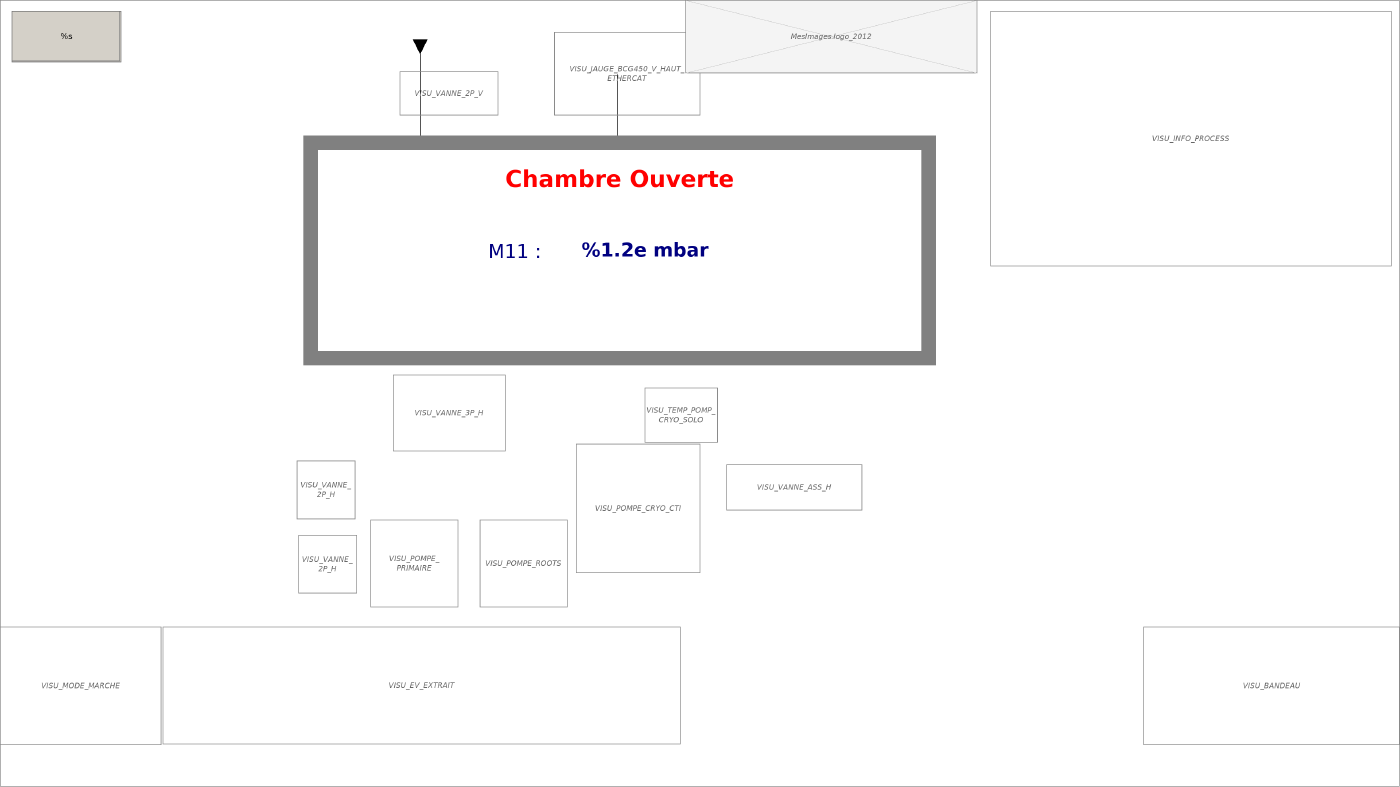
VISUALIZATION SYN_POMPAGE  // 1920x1080, background image fond_blanc_1280_1024
    Frame (223,860 710x161)
        shows VISU_EV_EXTRAIT()
    Frame (1568,860 352x162)
        shows VISU_BANDEAU(m_Input_MACHINE := Global_Variables.MACHINE)
    Frame (0,860 221x162)
        shows VISU_MODE_MARCHE(m_Input_MACHINE := .MACHINE)
    Button (16,15 150x70), "%s", text list: 'TextList_Navigation', text index: 1
        OnMouseClick: change screen: SYN_PROC
    Line (846,102) (846,217)
    Line (576,62) (576,216)
    RoundedRectangle (416,186 867x315)
    Frame (760,44 200x114)
        shows VISU_JAUGE_BCG450_V_HAUT_ETHERCAT(m_Input_JAUGE := PRG_POMPAGE.M11)
    Frame (548,98 135x60)
        shows VISU_VANNE_2P_V(m_Input_VANNE := PRG_POMPAGE.POMPAGE.VH11)
    Polygon (566,54) (586,54) (576,74)
    Rectangle (666,325 80x40), "M11 :"
    Rectangle (760,323 250x40), "%1.2e mbar", text variable: Global_Variables.PRG_POMPAGE.M11.STATE_Pression
    Label (669,214 362x63), "Chambre Ouverte", invisible if: PRG_POMPAGE.IN_FE11T
    Frame (1358,15 550x350), invisible if: NOT Global_Variables.MACHINE.STATE_Prod
        shows VISU_INFO_PROCESS()
    Polyline (458,705)
    Polyline (330,705)
    Polygon (337,745)
    Frame (407,632 80x80)
        shows VISU_VANNE_2P_H(m_Input_VANNE := PRG_POMPAGE.POMPAGE.VINT)
    Polyline (840,705)
    Frame (790,609 170x177)
        shows VISU_POMPE_CRYO_CTI(m_Input_POMPE := PRG_POMPAGE.POMPAGE.PS11, m_Input_COM := PRG_POMPAGE.COM_CRYOS, m_Input_Forcage := PRG_POMPAGE.POMPAGE.PS11.PRM_Forcage_Cryo_EXT)
    Polyline (553,751)
    Frame (884,532 100x75)
        shows VISU_TEMP_POMP_CRYO_SOLO(m_Input_CRYO := PRG_POMPAGE.COM_CRYOS, m_Input_PRG_POMPAGE := PRG_POMPAGE, m_Input_NumFrame_Manu := 2, m_Input_INDEX_CRYO := 1)
    Rectangle (170,643 200x30), text list: 'TextList_Pompage', text index: 0
    Polyline (458,664)
    Frame (508,713 120x120)
        shows VISU_POMPE_PRIMAIRE(m_Input_POMPE := PRG_POMPAGE.POMPAGE.PP11)
    Frame (658,713 120x120)
        shows VISU_POMPE_ROOTS(m_Input_POMPE := PRG_POMPAGE.POMPAGE.PR11)
    Frame (409,734 80x80)
        shows VISU_VANNE_2P_H(m_Input_VANNE := PRG_POMPAGE.POMPAGE.VN2PP11)
    Polygon (337,745)
    Image (940,0 400x100), image: MesImages.logo_2012
    Frame (539,514 154x105)
        shows VISU_VANNE_3P_H(m_Input_Vanne := PRG_POMPAGE.POMPAGE.VP11)
    Frame (996,637 186x63)
        shows VISU_VANNE_ASS_H(m_Input_VANNE := PRG_POMPAGE.POMPAGE.VS11, m_Input_NumFrame_Manu := 3)
END_VISUALIZATION

(* stored: Version 1.1.0.1, ProductVersion 3.1.4026.18
   Visu SYN_POMPAGE: Id {cb30cb57-0cb9-405d-ba2f-650bb21968ed} *)
